ABB RAPID module: INF_L.mod

MODULE INF_L
  ! Network configuration
  PERS string ipController:="192.168.125.1";
  PERS num motionPortR:=5000;
  PERS num loggerPortR:=5001;
  PERS num motionPortL:=5002;
  PERS num loggerPortL:=5003;
  PERS num infoPortR:=5004;
  PERS num infoPortL:=5005;
  PERS num loggerWaitTime:=0.1;

  ! Frame configuration
  PERS tooldata currentToolL:=[TRUE,[[0,0,130],[1,0,0,0]],[0.262,[7.8,11.9,50.7],[1,0,0,0],0.00022,0.00024,9E-05]];
  PERS wobjdata currentWobjL:=[FALSE,TRUE,"",[[0,0,0],[1,0,0,0]],[[0,0,0],[1,0,0,0]]];
  PERS speeddata currentSpeedL:=[50,10,5000,1000];
  PERS zonedata currentZoneL:=[FALSE,0.3,0.3,0.3,0.03,0.3,0.03];
  PERS tooldata currentToolR:=[TRUE,[[0,0,150],[1,0,0,0]],[0.262,[7.8,11.9,50.7],[1,0,0,0],0.00022,0.00024,9E-05]];
  PERS wobjdata currentWobjR:=[FALSE,TRUE,"",[[0,0,0],[1,0,0,0]],[[0,0,0],[1,0,0,0]]];
  PERS speeddata currentSpeedR:=[50,10,5000,1000];
  PERS zonedata currentZoneR:=[FALSE,0.3,0.3,0.3,0.03,0.3,0.03];

  ! Clock sync
  PERS bool startInfoL;
  PERS bool startLoggerL;
  PERS bool startMotionL;

  ! Mutex for frame modification
  PERS bool frameMutexL;

  ! Communication vars
  VAR socketdev clientSocket;
  VAR socketdev serverSocket;

  ! Vars for command parsing
  VAR num instructionCode;
  VAR string idCode;
  VAR num params{10};
  VAR num specialParams{5};
  VAR num nParams;

  ! External axis position variables
  VAR extjoint externalAxis;

  ! Error Handler
  VAR errnum ikErr;

  ! Upper and lower joint bounds, in degrees
  VAR num upper_joint_limits{7};
  VAR num lower_joint_limits{7};

  ! Inverse and forward kinematic results
  VAR jointtarget ikResult;
  VAR robtarget fkResult;

  ! Connection status
  VAR bool connected;        ! Client connected
  VAR bool reconnected;      ! Reconnection during the iteration

  ! Possible answers to controller
  VAR num ok;
  CONST num SERVER_BAD_MSG:=0;
  CONST num SERVER_OK:=1;
  CONST num SERVER_COLLISION:=2;
  CONST num SERVER_BAD_IK:=3;
  CONST num SERVER_BAD_FK:=4;

  ! Other variables
  VAR string receivedString;
  VAR string sendString;
  VAR string addString;
  VAR robtarget cartesianPose;
  VAR jointtarget jointsPose;
  VAR bool move;
  VAR clock timer;
  VAR bool isHandCalibrated;
  VAR num handSpeed;
  VAR num handPosition;

  ! Handshake between server and client:
  ! - Creates socket.
  ! - Waits for incoming TCP connection.
  PROC ConnectServer()
    VAR string clientIP;
    SocketCreate serverSocket;
    SocketBind serverSocket, ipController, infoPortL;
    SocketListen serverSocket;
    WHILE SocketGetStatus(clientSocket)<>SOCKET_CONNECTED DO
      SocketAccept serverSocket, clientSocket \ClientAddress:=clientIP \Time:=WAIT_MAX;
      IF SocketGetStatus(clientSocket)<>SOCKET_CONNECTED THEN
        TPWrite "Problem serving a connection. Try reconnecting.";
      ENDIF
      ! Wait 0.5 seconds for the next reconnection
      WaitTime 0.5;
    ENDWHILE
    TPWrite "Connected to "+clientIP+":"+NumToStr(infoPortL, 0);
    connected:=TRUE;
  ENDPROC

  ! Method to parse the message received from a PC through the socket
  ! Loads values on:
  ! - instructionCode.
  ! - idCode: 3 digit identifier of the command.
  ! - nParams: Number of received parameters.
  ! - params{nParams}: Vector of received params.
  PROC ParseMsg(string msg)
    VAR bool auxOk;
    VAR num ind:=1;
    VAR num newInd;
    VAR num length;
    VAR num indParam:=1;
    VAR string subString;
    VAR bool end:=FALSE;

    length:=StrMatch(msg,1,"#");
    IF length>StrLen(msg) THEN
      !Corrupt message
      nParams:=-1;
    ELSE
      ! Find Instruction code
      newInd:=StrMatch(msg,ind," ")+1;
      subString:=StrPart(msg,ind,newInd-ind-1);
      auxOk:=StrToVal(subString,instructionCode);
      IF auxOk=FALSE THEN
        !Corrupt instruction code
        nParams:=-1;
      ELSE
        ind:=newInd;

        !Find Id Code
        newInd:=StrMatch(msg,ind," ")+1;
        idCode:=StrPart(msg,ind,newInd-ind-1);
        ind:=newInd;

        !Set of parameters (maximum of 8)
        WHILE end=FALSE DO
          newInd:=StrMatch(msg,ind," ")+1;
          IF newInd>length THEN
            end:=TRUE;
          ELSE
            subString:=StrPart(msg,ind,newInd-ind-1);
            auxOk:=StrToVal(subString,params{indParam});
            indParam:=indParam+1;
            ind:=newInd;
          ENDIF
        ENDWHILE
        nParams:=indParam-1;
      ENDIF
    ENDIF
  ENDPROC

  ! Gets joint limits so they can be used later
  PROC ReadJointLimits()
    VAR string path;

    ! Get all of the joint bounds for later use
    FOR i FROM 1 TO 7 DO
      path:="MOC/ARM/rob_L_"+NumToStr(i,0);
      ReadCfgData path,"upper_joint_bound",upper_joint_limits{i};
      ReadCfgData path,"lower_joint_bound",lower_joint_limits{i};

      ! The joint limits are in radians, so convert these to degrees
      upper_joint_limits{i}:=upper_joint_limits{i}*180.0/pi;
      lower_joint_limits{i}:=lower_joint_limits{i}*180.0/pi;
    ENDFOR
  ENDPROC


  PROC main()
    ! Initially, we are not changing the frame
    frameMutexL:=FALSE;

    ! Gets joint limits so they can be used later
    ReadJointLimits;

    ! Wait until all tasks are ready
    WaitUntil startLoggerL \PollRate:=0.01;
    WaitUntil startMotionL \PollRate:=0.01;
    startInfoL:=TRUE;
    ClkStart timer;

    ! Socket connection
    ConnectServer;

    ! Infinite loop to serve commands
    WHILE TRUE DO
      ! Initialization of program flow variables
      ok:=SERVER_OK;
      reconnected:=FALSE;
      addString:="";

      ! Receive a command
      SocketReceive clientSocket \Str:=receivedString \Time:=WAIT_MAX;
      ParseMsg receivedString;

      ! Execution of the command
      TEST instructionCode
      CASE 0:
        ! Ping
        IF nParams=0 THEN
            ok:=SERVER_OK;
        ELSE
            ok:=SERVER_BAD_MSG;
        ENDIF


      CASE 3:
        ! GetCartesian
        IF nParams=0 THEN
          ! Read cartesian pose
          cartesianPose:=CRobT(\Tool:=currentToolL \WObj:=currentWobjL);

          ! Prepare string to send
          addString:=NumToStr(cartesianPose.trans.x,2)+" ";
          addString:=addString+NumToStr(cartesianPose.trans.y,2)+" ";
          addString:=addString+NumToStr(cartesianPose.trans.z,2)+" ";
          addString:=addString+NumToStr(cartesianPose.rot.q1,4)+" ";
          addString:=addString+NumToStr(cartesianPose.rot.q2,4)+" ";
          addString:=addString+NumToStr(cartesianPose.rot.q3,4)+" ";
          addString:=addString+NumToStr(cartesianPose.rot.q4,4);
          ok:=SERVER_OK;
        ELSE
          ok:=SERVER_BAD_MSG;
        ENDIF


      CASE 4:
        ! GetJoints
        IF nParams=0 THEN
          ! Read joint coordinates
          jointsPose:=CJointT();

          ! Prepare string to send
          addString:=NumToStr(jointsPose.robax.rax_1,2)+" ";
          addString:=addString+NumToStr(jointsPose.robax.rax_2,2)+" ";
          addString:=addString+NumToStr(jointsPose.robax.rax_3,2)+" ";
          addString:=addString+NumToStr(jointsPose.robax.rax_4,2)+" ";
          addString:=addString+NumToStr(jointsPose.robax.rax_5,2)+" ";
          addString:=addString+NumToStr(jointsPose.robax.rax_6,2)+" ";
          addString:=addString+NumToStr(jointsPose.extax.eax_a,2);
          !End of string
          ok:=SERVER_OK;
        ELSE
          ok:=SERVER_BAD_MSG;
        ENDIF


      CASE 6:
        ! SetTool
        IF nParams=7 THEN
          ! Wait until frame is not being used (e.g. by logger) and then block it
          WHILE (frameMutexL) DO
          ENDWHILE
          frameMutexL:=TRUE;

          ! Set new values and unblock frame again
          currentToolL.tframe.trans.x:=params{1};
          currentToolL.tframe.trans.y:=params{2};
          currentToolL.tframe.trans.z:=params{3};
          currentToolL.tframe.rot.q1:=params{4};
          currentToolL.tframe.rot.q2:=params{5};
          currentToolL.tframe.rot.q3:=params{6};
          currentToolL.tframe.rot.q4:=params{7};
          frameMutexL:=FALSE;
          ok:=SERVER_OK;
        ELSE
          ok:=SERVER_BAD_MSG;
        ENDIF


      CASE 7:
        ! SetWorkObject
        IF nParams=7 THEN
          ! Wait until frame is not being used (e.g. by logger) and then block it
          WHILE (frameMutexL) DO
          ENDWHILE
          frameMutexL:=TRUE;
          currentWobjL.oframe.trans.x:=params{1};
          currentWobjL.oframe.trans.y:=params{2};
          currentWobjL.oframe.trans.z:=params{3};
          currentWobjL.oframe.rot.q1:=params{4};
          currentWobjL.oframe.rot.q2:=params{5};
          currentWobjL.oframe.rot.q3:=params{6};
          currentWobjL.oframe.rot.q4:=params{7};
          frameMutexL:=FALSE;
          ok:=SERVER_OK;
        ELSE
          ok:=SERVER_BAD_MSG;
        ENDIF


      CASE 8:
        ! SetMaxSpeed
        IF nParams=2 THEN
          currentSpeedL.v_tcp:=params{1};
          currentSpeedL.v_ori:=params{2};
          ok:=SERVER_OK;
        ELSE
          ok:=SERVER_BAD_MSG;
        ENDIF


      CASE 9:
        ! SetZone
        IF nParams=4 THEN
          IF params{1}=1 THEN
            currentZoneL.finep:=TRUE;
            currentZoneL.pzone_tcp:=0.0;
            currentZoneL.pzone_ori:=0.0;
            currentZoneL.zone_ori:=0.0;
          ELSE
            currentZoneL.finep:=FALSE;
            currentZoneL.pzone_tcp:=params{2};
            currentZoneL.pzone_ori:=params{3};
            currentZoneL.zone_ori:=params{4};
          ENDIF
          ok:=SERVER_OK;
        ELSE
          ok:=SERVER_BAD_MSG;
        ENDIF

      CASE 10:
        ! GetRobotAngle
        IF nParams=0 THEN
            cartesianPose:=CRobT(\Tool:=currentToolL \WObj:=currentWobjL);
            addString:=NumToStr(cartesianPose.extax.eax_a,2);
            ok:=SERVER_OK;
        ELSE
            ok:=SERVER_BAD_MSG;
        ENDIF


      CASE 12:
        ! GetIK
        IF nParams=8 THEN
          ! First, let's make sure the quaternion is normalized
          IF Abs(1.0-Sqrt(params{4}*params{4}+params{5}*params{5}+params{6}*params{6}+params{7}*params{7}))>0.001 THEN
            ! If not, then we cannot find the inverse kinematics for this pose
            ok:=SERVER_BAD_IK;
          ELSE
            ! Otherwise, let's normalize our quaternion
            cartesianPose:=[[params{1},params{2},params{3}],
                NOrient([params{4},params{5},params{6},params{7}]),
                [-1, -1, 0, 11],
                [params{8},9E9,9E9,9E9,9E9,9E9]];
            ok:=SERVER_OK;

            ! Now calculate the joint angles, keeping in mind that if we specified an
            ! impossible configuration, this will generate an error (See error handler below)
            ikResult:=CalcJointT(cartesianPose, currentToolL, \WObj:=currentWobjL, \ErrorNumber:=ikErr);

            ! Store our result in a string to return to the user
            addString:=NumToStr(ikResult.robax.rax_1,2)+" ";
            addString:=addString+NumToStr(ikResult.robax.rax_2,2)+" ";
            addString:=addString+NumToStr(ikResult.robax.rax_3,2)+" ";
            addString:=addString+NumToStr(ikResult.robax.rax_4,2)+" ";
            addString:=addString+NumToStr(ikResult.robax.rax_5,2)+" ";
            addString:=addString+NumToStr(ikResult.robax.rax_6,2)+" ";
            addString:=addString+NumToStr(ikResult.extax.eax_a,2)+" ";
            addString:=addString+NumToStr(ikErr,2);
            !End of string
          ENDIF
        ELSE
          ok:=SERVER_BAD_MSG;
        ENDIF


      CASE 13:
        ! GetFK
        IF nParams=7 THEN
          ok:=SERVER_OK;

          ! First, let's make sure the specified joint angles are within range
          FOR i FROM 1 TO 7 DO
            IF params{i}>upper_joint_limits{i}OR params{i}<lower_joint_limits{i} THEN
              ! If not, then we'll tell the user that their forward kinematics are invalid
              ok:=SERVER_BAD_FK;
            ENDIF
          ENDFOR

          ! If our joints are within limits, then let's carry on
          IF ok=SERVER_OK THEN
            ! Create a joint target, and then calculate the corresponding cartesian pose
            jointsPose:=[[params{1},params{2},params{3},params{4},params{5},params{6}],
                    [params{7},9E9,9E9,9E9,9E9,9E9]];
            fkResult:=CalcRobT(jointsPose,currentToolL,\WObj:=currentWobjL);

            ! Now add this pose to our return string
            addString:=NumToStr(fkResult.trans.x,2)+" ";
            addString:=addString+NumToStr(fkResult.trans.y,2)+" ";
            addString:=addString+NumToStr(fkResult.trans.z,2)+" ";
            addString:=addString+NumToStr(fkResult.rot.q1,4)+" ";
            addString:=addString+NumToStr(fkResult.rot.q2,4)+" ";
            addString:=addString+NumToStr(fkResult.rot.q3,4)+" ";
            addString:=addString+NumToStr(fkResult.rot.q4,4);
          ENDIF
        ELSE
          ok:=SERVER_BAD_MSG;
        ENDIF


      CASE 14:
        ! SetInertia
        IF nParams=7 THEN
          currentToolL.tload.mass:=params{1};
          currentToolL.tload.cog.x:=params{2};
          currentToolL.tload.cog.y:=params{3};
          currentToolL.tload.cog.z:=params{4};
          currentToolL.tload.ix:=params{5};
          currentToolL.tload.iy:=params{6};
          currentToolL.tload.iz:=params{7};
          currentToolL.tload.aom.q1:=1.0;
          currentToolL.tload.aom.q2:=0.0;
          currentToolL.tload.aom.q3:=0.0;
          currentToolL.tload.aom.q4:=0.0;
          ok:=SERVER_OK;
        ELSE
          ok:=SERVER_BAD_MSG;
        ENDIF


      CASE 23:
        ! Check if gripper is calibrated
        IF nParams=0 THEN
          isHandCalibrated := Hand_IsCalibrated();
          IF isHandCalibrated THEN
              addString:=NumToStr(1,2);
          ELSE
              addString:=NumToStr(0,2);
          ENDIF
          ok:=SERVER_OK;
        ELSE
          ok:=SERVER_BAD_MSG;
        ENDIF


      CASE 24:
        ! Get current gripper position
        IF nParams=0 THEN
          handPosition := Hand_GetActualPos();
          addString:=NumToStr(handPosition,2);
          ok:=SERVER_OK;
        ELSE
          ok:=SERVER_BAD_MSG;
        ENDIF


      CASE 99:
        ! CloseServer
        IF nParams=0 THEN
          TPWrite "Connection closed by client.";
          connected:=FALSE;
          ! Closing the server
          SocketClose clientSocket;
          SocketClose serverSocket;

          ! Reinitiate the server
          ConnectServer;
          connected:=TRUE;
          reconnected:=TRUE;
          ok:=SERVER_OK;
        ELSE
          ok:=SERVER_BAD_MSG;
        ENDIF


      DEFAULT:
        TPWrite "Illegal instruction code";
        ok:=SERVER_BAD_MSG;
      ENDTEST

      ! Finally we compose the acknowledge string to send back to the client
      abort:
      IF connected=TRUE THEN
        IF reconnected=FALSE THEN
          sendString:=NumToStr(instructionCode,0);
          sendString:=sendString+" "+idCode;
          sendString:=sendString+" "+NumToStr(ok,0);
          sendString:=sendString+" "+NumToStr(ClkRead(timer),2);
          sendString:=sendString+" "+addString+ByteToStr(10\Char);
          SocketSend clientSocket\Str:=sendString;
        ENDIF
      ENDIF
    ENDWHILE
  ERROR (LONG_JMP_ALL_ERR)
    TEST ERRNO
    CASE ERR_SOCK_CLOSED:
      TPWrite "Connection closed by client.";
      connected:=FALSE;

      ! Closing the server
      SocketClose clientSocket;
      SocketClose serverSocket;

      ! Reinitiate the server
      ConnectServer;
      reconnected:=TRUE;
      connected:=TRUE;
      TRYNEXT;

    CASE ERR_ROBLIMIT:
      ! Out of reach cartesian target.
      ok:=SERVER_BAD_IK;

      ! Skip the instruction computing the IK that caused the error
      TRYNEXT;

    DEFAULT:
      TPWrite "Unknown error (" +NumtoStr(ERRNO,0)+ "). Restarting.";
      connected:=FALSE;
      ! Closing the server
      SocketClose clientSocket;
      SocketClose serverSocket;
      ! Reinitiate the server
      ConnectServer;
      reconnected:=TRUE;
      connected:=TRUE;
      RETRY;
    ENDTEST
  ENDPROC
ENDMODULE
